// TIA Portal project "project_tia_portal" (V17)

(* hardware
DEVICE "S7-1500/ET200MP station_1"  S7-1500 station
   slot 0: "Rail_0"  Rack  6ES7 590-1***0-0AA0
   slot 1: "PLC_1"  CPU 1513-1 PN  6ES7 513-1AL01-0AB0  V2.6
      slot 3: "CPU display_1"  6ES7591-1AA00-0AA0
      slot 32768: "PROFINET interface_1"  X1
         slot 32769: "Port_1"  X1 P1
         slot 32770: "Port_2"  X1 P2
*)

// ===== PLC "PLC_1"  CPU 1513-1 PN =====

VAR_GLOBAL   // PLC tag table "Default tag table"
   "OPC_START" AT %I0.0 : Bool;
   "OPC_STOP" AT %I0.1 : Bool;
   "SISTEM" AT %M0.0 : Bool;
   "OPC_EMITTER" AT %Q0.0 : Bool;
   "OPC_LONG_BELT" AT %QD2 : Real;
   "OPC_CAPACITIVE_1" AT %I0.2 : Bool;
   "OPC_CAM" AT %QD6 : DInt;
   "OPC_PHOTOELECTRIC" AT %I0.3 : Bool;
   "OPC_GATE_1" AT %Q0.1 : Bool;
   "OPC_GATE_2" AT %Q0.2 : Bool;
   "OPC_PISTON_SENSOR" AT %I0.4 : Bool;
   "OPC_BELT_2" AT %Q0.3 : Bool;
   "OPC_PISTON" AT %QD10 : Real;
   "OPC_CAPACITIVE_2" AT %I0.5 : Bool;
   "ENABLE_BELT_2" AT %M0.5 : Bool;
   "OPC_GATE_FINALE" AT %Q0.4 : Bool;
   "OPC_CAPACITIVE_3" AT %I0.6 : Bool;
   "OPC_X_OUT" AT %QD14 : Real;
   "OPC_Y_OUT" AT %QD18 : Real;
   "OPC_Z_OUT" AT %QD22 : Real;
   "OPC_XY_MOVEMENT" AT %I0.7 : Bool;
   "OPC_Z_MOVEMENT" AT %I1.0 : Bool;
   "OPC_CONFIG" AT %I1.1 : Bool;
   "OPC_EMITTER_2" AT %Q0.5 : Bool;
   "OPC_X_IN" AT %ID2 : Real;
   "OPC_Y_IN" AT %ID6 : Real;
   "OPC_Z_IN" AT %ID10 : Real;
   "OPC_CLAW_BOX_DETECTED" AT %I1.2 : Bool;
   "OPC_CLAW" AT %Q0.6 : Bool;
   "OPC_BELT_LAST_1" AT %Q0.7 : Bool;
   "OPC_BELT_LAST_2" AT %Q1.0 : Bool;
END_VAR

DATA_BLOCK "IEC_Timer_0_DB"   // DB1
{ S7_Optimized_Access := 'TRUE' }
AUTHOR : Simatic
FAMILY : IEC
NAME : IEC_TMR
VERSION : 1.0
// stored: InstanceOfName IEC_TIMER
"IEC_TIMER"
BEGIN
END_DATA_BLOCK

DATA_BLOCK "IEC_Counter_0_DB"   // DB2
{ S7_Optimized_Access := 'TRUE' }
AUTHOR : Simatic
FAMILY : IEC
NAME : CNTR
VERSION : 1.0
// stored: InstanceOfName IEC_COUNTER
"IEC_COUNTER"
BEGIN
END_DATA_BLOCK

DATA_BLOCK "COORDS"   // DB3
{ S7_Optimized_Access := 'TRUE' }
VERSION : 0.1
   VAR
      BOX_X : Real;
      BOX_Y : Real;
      CODE : Int;
      X_LOW : Real;
      X_HIGH : Real;
      Y_LOW : Real;
      Y_HIGH : Real;
      Z_LOW : Real;
      Z_HIGH : Real;
      Y_FINALE : Real;
   END_VAR
BEGIN
END_DATA_BLOCK

DATA_BLOCK "CONFIG_VARS"   // DB7
{ S7_Optimized_Access := 'TRUE' }
VERSION : 0.1
   VAR
      MOVE_2_BOX : Bool;
      Y_POSITION_FINAL : Bool;
      EMITTER_CONFIG : Bool;
      Z_POSITION_FINALE : Bool;
      "COUNTER" : Int;
      TRIG_4_PY_INSTRUCTION : Bool;
      INSTRUCTION_2_PY : Bool;
      PY_RESPONSE : Bool;
      CONFIG_END : Bool;
      TRIG_N : Bool;
      INSTRUCTION_TRIG_N : Bool;
      GATE_FINALE : Bool;
      N_TRIG_FOR_EMITTER : Bool;
      FIRST_MOVE : Bool;
      SECOND_MOV : Bool;
      TRIG_4_MOVE : Bool;
      TRIG_4_2ND_MOVE : Bool;
      TRIG_4_CLAW : Bool;
      TRIG_4_DROP : Bool;
      TRIG_4_RSTART : Bool;
      N_TRIG_FIRST_MOV : Bool;
      N_TRIG_SISTEM : Bool;
   END_VAR
BEGIN
END_DATA_BLOCK

DATA_BLOCK "PRINCIPAL"   // DB8
{ S7_Optimized_Access := 'TRUE' }
VERSION : 0.1
   VAR
      "2_UNITS" : Int;
      N_TRIG_2_UDS : Bool;
      P_TRIG_LONG_BELT : Bool;
      N_TRIG_LONG_BELT : Bool;
      TRIG : Bool;
   END_VAR
BEGIN
END_DATA_BLOCK

DATA_BLOCK "Emitters"   // DB11
{ S7_Optimized_Access := 'TRUE' }
VERSION : 0.1
   VAR
      Trig_1 : Bool;
      Trig_2 : Bool;
      Trig_3 : Bool;
      Trig_4 : Bool;
      Trig_5 : Bool;
   END_VAR
BEGIN
END_DATA_BLOCK

// folder: System blocks/Program resources

DATA_BLOCK "IEC_Timer_0_DB_1"   // DB4
{ S7_Optimized_Access := 'TRUE' }
AUTHOR : Simatic
FAMILY : IEC
NAME : IEC_TMR
VERSION : 1.0
// stored: InstanceOfName IEC_TIMER
"IEC_TIMER"
BEGIN
END_DATA_BLOCK

DATA_BLOCK "IEC_Timer_0_DB_2"   // DB5
{ S7_Optimized_Access := 'TRUE' }
AUTHOR : Simatic
FAMILY : IEC
NAME : IEC_TMR
VERSION : 1.0
// stored: InstanceOfName IEC_TIMER
"IEC_TIMER"
BEGIN
END_DATA_BLOCK

DATA_BLOCK "IEC_Timer_0_DB_3"   // DB6
{ S7_Optimized_Access := 'TRUE' }
AUTHOR : Simatic
FAMILY : IEC
NAME : IEC_TMR
VERSION : 1.0
// stored: InstanceOfName IEC_TIMER
"IEC_TIMER"
BEGIN
END_DATA_BLOCK

DATA_BLOCK "IEC_Timer_0_DB_4"   // DB9
{ S7_Optimized_Access := 'TRUE' }
AUTHOR : Simatic
FAMILY : IEC
NAME : IEC_TMR
VERSION : 1.0
// stored: InstanceOfName IEC_TIMER
"IEC_TIMER"
BEGIN
END_DATA_BLOCK

DATA_BLOCK "IEC_Timer_0_DB_5"   // DB10
{ S7_Optimized_Access := 'TRUE' }
AUTHOR : Simatic
FAMILY : IEC
NAME : IEC_TMR
VERSION : 1.0
// stored: InstanceOfName IEC_TIMER
"IEC_TIMER"
BEGIN
END_DATA_BLOCK

// folder: (top level)

FUNCTION "PICK_PLACE" : Void   // FC2, LAD
{ S7_Optimized_Access := 'TRUE' }
VERSION : 0.1
   VAR_TEMP
      EMITTER_CONFIG : Bool;
      EMITTER_CONFIG_1 : Bool;
      EMITTER_CONFIG_2 : Bool;
   END_VAR
   VAR_TEMP   // added for the SCL form of the ladder/FBD networks
      _w1 : Bool;
      _w2 : Bool;
      _w3 : Bool;
      _w4 : Bool;
      _w5 : Bool;
      _w6 : Bool;
   END_VAR
BEGIN

REGION Network 1
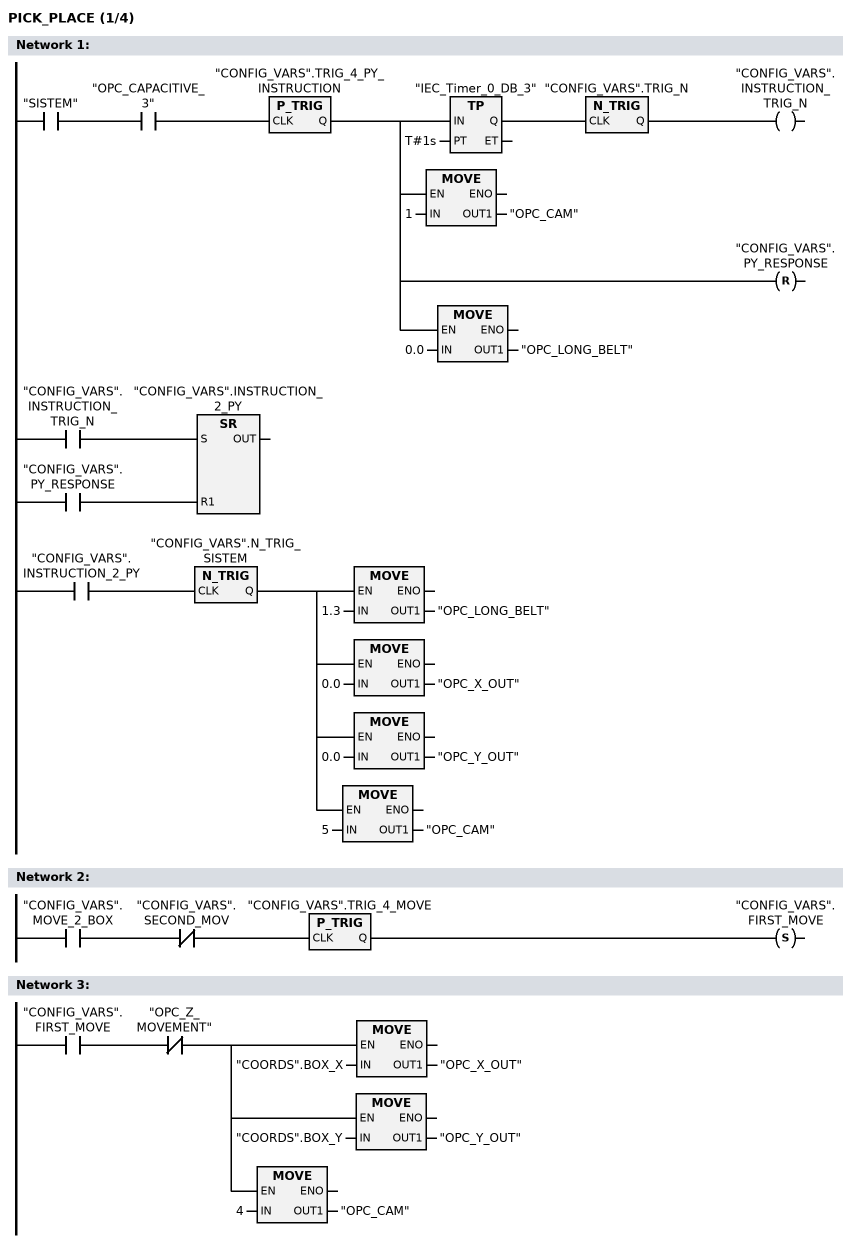
   #_w1 := "SISTEM" AND "OPC_CAPACITIVE_3";
   #_w2 := #_w1 AND NOT "CONFIG_VARS".TRIG_4_PY_INSTRUCTION;   // rising edge
   "CONFIG_VARS".TRIG_4_PY_INSTRUCTION := #_w1;
   "IEC_Timer_0_DB_3".TP(IN := #_w2, PT := T#1s);
   #_w3 := NOT "IEC_Timer_0_DB_3".Q AND "CONFIG_VARS".TRIG_N;   // falling edge
   "CONFIG_VARS".TRIG_N := "IEC_Timer_0_DB_3".Q;
   "CONFIG_VARS".INSTRUCTION_TRIG_N := #_w3;
   IF #_w2 THEN
       "OPC_CAM" := 1;
       "CONFIG_VARS".PY_RESPONSE := FALSE;
       "OPC_LONG_BELT" := 0.0;
   END_IF;
   IF "CONFIG_VARS".INSTRUCTION_TRIG_N THEN
       "CONFIG_VARS".INSTRUCTION_2_PY := TRUE;   // SR flip-flop
   END_IF;
   IF "CONFIG_VARS".PY_RESPONSE THEN "CONFIG_VARS".INSTRUCTION_2_PY := FALSE; END_IF;
   #_w4 := NOT "CONFIG_VARS".INSTRUCTION_2_PY AND "CONFIG_VARS".N_TRIG_SISTEM;   // falling edge
   "CONFIG_VARS".N_TRIG_SISTEM := "CONFIG_VARS".INSTRUCTION_2_PY;
   IF #_w4 THEN
       "OPC_LONG_BELT" := 1.3;
       "OPC_X_OUT" := 0.0;
       "OPC_Y_OUT" := 0.0;
       "OPC_CAM" := 5;
   END_IF;
END_REGION

REGION Network 2
   RUNG wire#powerrail
      Contact( "CONFIG_VARS".MOVE_2_BOX )
      I_Contact( "CONFIG_VARS".SECOND_MOV )
      P_Trig( "CONFIG_VARS".TRIG_4_MOVE )
      S_Coil( "CONFIG_VARS".FIRST_MOVE )
   END_RUNG
   // the same network as SCL:
   #_w1 := "CONFIG_VARS".MOVE_2_BOX AND NOT "CONFIG_VARS".SECOND_MOV;
   #_w2 := #_w1 AND NOT "CONFIG_VARS".TRIG_4_MOVE;   // rising edge
   "CONFIG_VARS".TRIG_4_MOVE := #_w1;
   IF #_w2 THEN "CONFIG_VARS".FIRST_MOVE := TRUE; END_IF;
END_REGION

REGION Network 3
   RUNG wire#powerrail
      Contact( "CONFIG_VARS".FIRST_MOVE )
      I_Contact( "OPC_Z_MOVEMENT" )
      wire#w1
      Move(in := "COORDS".BOX_X, out1 => "OPC_X_OUT")
   END_RUNG
   RUNG wire#w1
      Move(in := "COORDS".BOX_Y, out1 => "OPC_Y_OUT")
   END_RUNG
   RUNG wire#w1
      Move(in := 4, out1 => "OPC_CAM")
   END_RUNG
   // the same network as SCL:
   IF "CONFIG_VARS".FIRST_MOVE AND NOT "OPC_Z_MOVEMENT" THEN
       "OPC_X_OUT" := "COORDS".BOX_X;
       "OPC_Y_OUT" := "COORDS".BOX_Y;
       "OPC_CAM" := 4;
   END_IF;
END_REGION

REGION Network 4
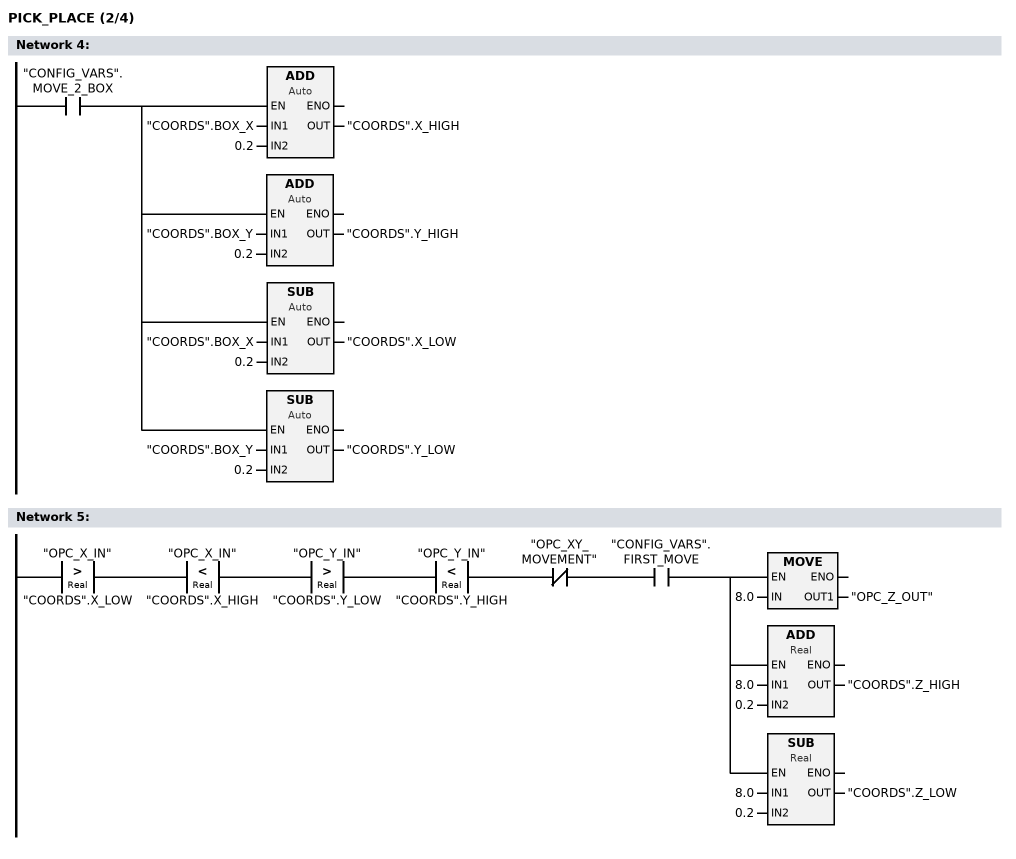
   RUNG wire#powerrail
      Contact( "CONFIG_VARS".MOVE_2_BOX )
      wire#w1
      Add(in1 := "COORDS".BOX_X, in2 := 0.2, out => "COORDS".X_HIGH)
   END_RUNG
   RUNG wire#w1
      Add(in1 := "COORDS".BOX_Y, in2 := 0.2, out => "COORDS".Y_HIGH)
   END_RUNG
   RUNG wire#w1
      Sub(in1 := "COORDS".BOX_X, in2 := 0.2, out => "COORDS".X_LOW)
   END_RUNG
   RUNG wire#w1
      Sub(in1 := "COORDS".BOX_Y, in2 := 0.2, out => "COORDS".Y_LOW)
   END_RUNG
   // the same network as SCL:
   IF "CONFIG_VARS".MOVE_2_BOX THEN
       "COORDS".X_HIGH := "COORDS".BOX_X + 0.2;
       "COORDS".Y_HIGH := "COORDS".BOX_Y + 0.2;
       "COORDS".X_LOW := "COORDS".BOX_X - 0.2;
       "COORDS".Y_LOW := "COORDS".BOX_Y - 0.2;
   END_IF;
END_REGION

REGION Network 5
   RUNG wire#powerrail
      { S7_Templates := "SrcType := Real" } GT_Contact(in1 := "OPC_X_IN", in2 := "COORDS".X_LOW)
      { S7_Templates := "SrcType := Real" } LT_Contact(in1 := "OPC_X_IN", in2 := "COORDS".X_HIGH)
      { S7_Templates := "SrcType := Real" } GT_Contact(in1 := "OPC_Y_IN", in2 := "COORDS".Y_LOW)
      { S7_Templates := "SrcType := Real" } LT_Contact(in1 := "OPC_Y_IN", in2 := "COORDS".Y_HIGH)
      I_Contact( "OPC_XY_MOVEMENT" )
      Contact( "CONFIG_VARS".FIRST_MOVE )
      wire#w1
      Move(in := 8.0, out1 => "OPC_Z_OUT")
   END_RUNG
   RUNG wire#w1
      { S7_Templates := "SrcType := Real" } Add(in1 := 8.0, in2 := 0.2, out => "COORDS".Z_HIGH)
   END_RUNG
   RUNG wire#w1
      { S7_Templates := "SrcType := Real" } Sub(in1 := 8.0, in2 := 0.2, out => "COORDS".Z_LOW)
   END_RUNG
   // the same network as SCL:
   IF ("OPC_X_IN" > "COORDS".X_LOW) AND ("OPC_X_IN" < "COORDS".X_HIGH) AND ("OPC_Y_IN" > "COORDS".Y_LOW) AND ("OPC_Y_IN" < "COORDS".Y_HIGH) AND NOT "OPC_XY_MOVEMENT" AND "CONFIG_VARS".FIRST_MOVE THEN
       "OPC_Z_OUT" := 8.0;
       "COORDS".Z_HIGH := 8.0 + 0.2;
       "COORDS".Z_LOW := 8.0 - 0.2;
   END_IF;
END_REGION

REGION Network 6
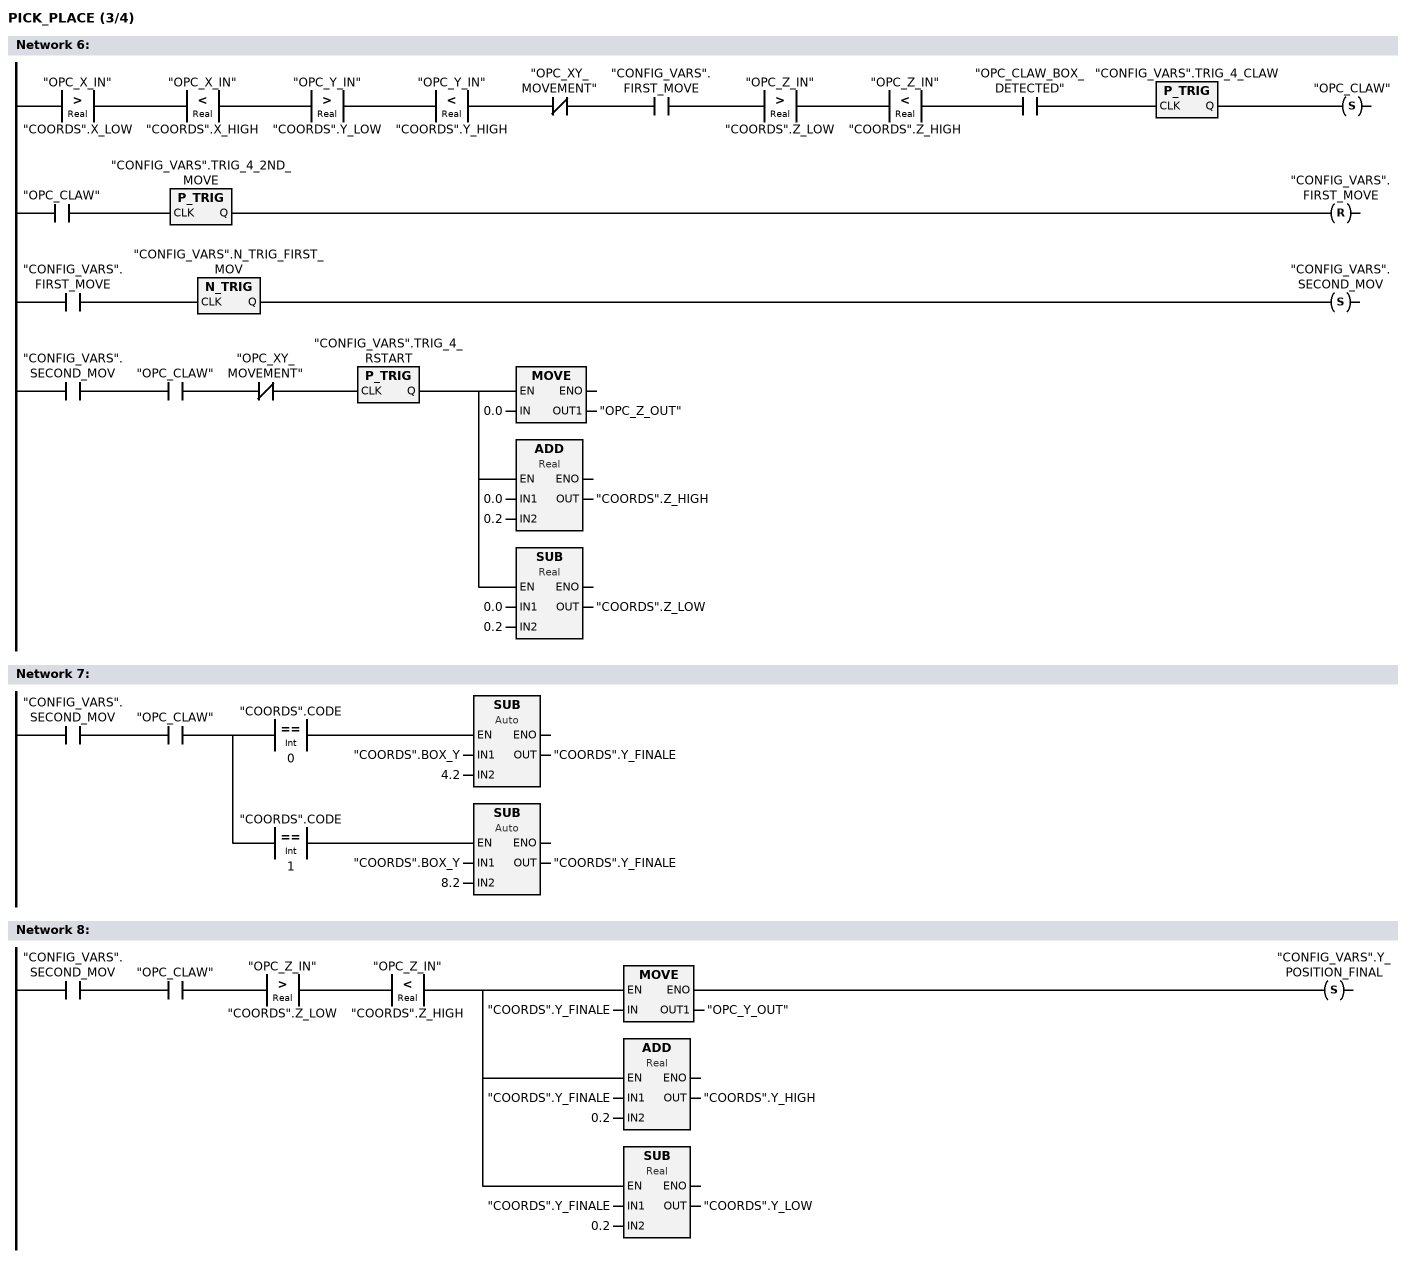
   RUNG wire#powerrail
      { S7_Templates := "SrcType := Real" } GT_Contact(in1 := "OPC_X_IN", in2 := "COORDS".X_LOW)
      { S7_Templates := "SrcType := Real" } LT_Contact(in1 := "OPC_X_IN", in2 := "COORDS".X_HIGH)
      { S7_Templates := "SrcType := Real" } GT_Contact(in1 := "OPC_Y_IN", in2 := "COORDS".Y_LOW)
      { S7_Templates := "SrcType := Real" } LT_Contact(in1 := "OPC_Y_IN", in2 := "COORDS".Y_HIGH)
      I_Contact( "OPC_XY_MOVEMENT" )
      Contact( "CONFIG_VARS".FIRST_MOVE )
      { S7_Templates := "SrcType := Real" } GT_Contact(in1 := "OPC_Z_IN", in2 := "COORDS".Z_LOW)
      { S7_Templates := "SrcType := Real" } LT_Contact(in1 := "OPC_Z_IN", in2 := "COORDS".Z_HIGH)
      Contact( "OPC_CLAW_BOX_DETECTED" )
      P_Trig( "CONFIG_VARS".TRIG_4_CLAW )
      S_Coil( "OPC_CLAW" )
   END_RUNG
   RUNG wire#powerrail
      Contact( "OPC_CLAW" )
      P_Trig( "CONFIG_VARS".TRIG_4_2ND_MOVE )
      R_Coil( "CONFIG_VARS".FIRST_MOVE )
   END_RUNG
   RUNG wire#powerrail
      Contact( "CONFIG_VARS".FIRST_MOVE )
      N_Trig( "CONFIG_VARS".N_TRIG_FIRST_MOV )
      S_Coil( "CONFIG_VARS".SECOND_MOV )
   END_RUNG
   RUNG wire#powerrail
      Contact( "CONFIG_VARS".SECOND_MOV )
      Contact( "OPC_CLAW" )
      I_Contact( "OPC_XY_MOVEMENT" )
      P_Trig( "CONFIG_VARS".TRIG_4_RSTART )
      wire#w1
      Move(in := 0.0, out1 => "OPC_Z_OUT")
   END_RUNG
   RUNG wire#w1
      { S7_Templates := "SrcType := Real" } Add(in1 := 0.0, in2 := 0.2, out => "COORDS".Z_HIGH)
   END_RUNG
   RUNG wire#w1
      { S7_Templates := "SrcType := Real" } Sub(in1 := 0.0, in2 := 0.2, out => "COORDS".Z_LOW)
   END_RUNG
   // the same network as SCL:
   #_w1 := ("OPC_X_IN" > "COORDS".X_LOW) AND ("OPC_X_IN" < "COORDS".X_HIGH) AND ("OPC_Y_IN" > "COORDS".Y_LOW) AND ("OPC_Y_IN" < "COORDS".Y_HIGH) AND NOT "OPC_XY_MOVEMENT" AND "CONFIG_VARS".FIRST_MOVE AND ("OPC_Z_IN" > "COORDS".Z_LOW) AND ("OPC_Z_IN" < "COORDS".Z_HIGH) AND "OPC_CLAW_BOX_DETECTED";
   #_w2 := #_w1 AND NOT "CONFIG_VARS".TRIG_4_CLAW;   // rising edge
   "CONFIG_VARS".TRIG_4_CLAW := #_w1;
   IF #_w2 THEN "OPC_CLAW" := TRUE; END_IF;
   #_w3 := "OPC_CLAW" AND NOT "CONFIG_VARS".TRIG_4_2ND_MOVE;   // rising edge
   "CONFIG_VARS".TRIG_4_2ND_MOVE := "OPC_CLAW";
   IF #_w3 THEN "CONFIG_VARS".FIRST_MOVE := FALSE; END_IF;
   #_w4 := NOT "CONFIG_VARS".FIRST_MOVE AND "CONFIG_VARS".N_TRIG_FIRST_MOV;   // falling edge
   "CONFIG_VARS".N_TRIG_FIRST_MOV := "CONFIG_VARS".FIRST_MOVE;
   IF #_w4 THEN "CONFIG_VARS".SECOND_MOV := TRUE; END_IF;
   #_w5 := "CONFIG_VARS".SECOND_MOV AND "OPC_CLAW" AND NOT "OPC_XY_MOVEMENT";
   #_w6 := #_w5 AND NOT "CONFIG_VARS".TRIG_4_RSTART;   // rising edge
   "CONFIG_VARS".TRIG_4_RSTART := #_w5;
   IF #_w6 THEN
       "OPC_Z_OUT" := 0.0;
       "COORDS".Z_HIGH := 0.0 + 0.2;
       "COORDS".Z_LOW := 0.0 - 0.2;
   END_IF;
END_REGION

REGION Network 7
   RUNG wire#powerrail
      Contact( "CONFIG_VARS".SECOND_MOV )
      Contact( "OPC_CLAW" )
      wire#w1
      { S7_Templates := "SrcType := Int" } EQ_Contact(in1 := "COORDS".CODE, in2 := 0)
      Sub(in1 := "COORDS".BOX_Y, in2 := 4.2, out => "COORDS".Y_FINALE)
   END_RUNG
   RUNG wire#w1
      { S7_Templates := "SrcType := Int" } EQ_Contact(in1 := "COORDS".CODE, in2 := 1)
      Sub(in1 := "COORDS".BOX_Y, in2 := 8.2, out => "COORDS".Y_FINALE)
   END_RUNG
   // the same network as SCL:
   #_w1 := "CONFIG_VARS".SECOND_MOV AND "OPC_CLAW";
   IF #_w1 AND ("COORDS".CODE = 0) THEN "COORDS".Y_FINALE := "COORDS".BOX_Y - 4.2; END_IF;
   IF #_w1 AND ("COORDS".CODE = 1) THEN "COORDS".Y_FINALE := "COORDS".BOX_Y - 8.2; END_IF;
END_REGION

REGION Network 8
   RUNG wire#powerrail
      Contact( "CONFIG_VARS".SECOND_MOV )
      Contact( "OPC_CLAW" )
      { S7_Templates := "SrcType := Real" } GT_Contact(in1 := "OPC_Z_IN", in2 := "COORDS".Z_LOW)
      { S7_Templates := "SrcType := Real" } LT_Contact(in1 := "OPC_Z_IN", in2 := "COORDS".Z_HIGH)
      wire#w1
      Move(in := "COORDS".Y_FINALE, out1 => "OPC_Y_OUT")
      S_Coil( "CONFIG_VARS".Y_POSITION_FINAL )
   END_RUNG
   RUNG wire#w1
      { S7_Templates := "SrcType := Real" } Add(in1 := "COORDS".Y_FINALE, in2 := 0.2, out => "COORDS".Y_HIGH)
   END_RUNG
   RUNG wire#w1
      { S7_Templates := "SrcType := Real" } Sub(in1 := "COORDS".Y_FINALE, in2 := 0.2, out => "COORDS".Y_LOW)
   END_RUNG
   // the same network as SCL:
   IF "CONFIG_VARS".SECOND_MOV AND "OPC_CLAW" AND ("OPC_Z_IN" > "COORDS".Z_LOW) AND ("OPC_Z_IN" < "COORDS".Z_HIGH) THEN
       "OPC_Y_OUT" := "COORDS".Y_FINALE;
       "CONFIG_VARS".Y_POSITION_FINAL := TRUE;
       "COORDS".Y_HIGH := "COORDS".Y_FINALE + 0.2;
       "COORDS".Y_LOW := "COORDS".Y_FINALE - 0.2;
   END_IF;
END_REGION

REGION Network 9
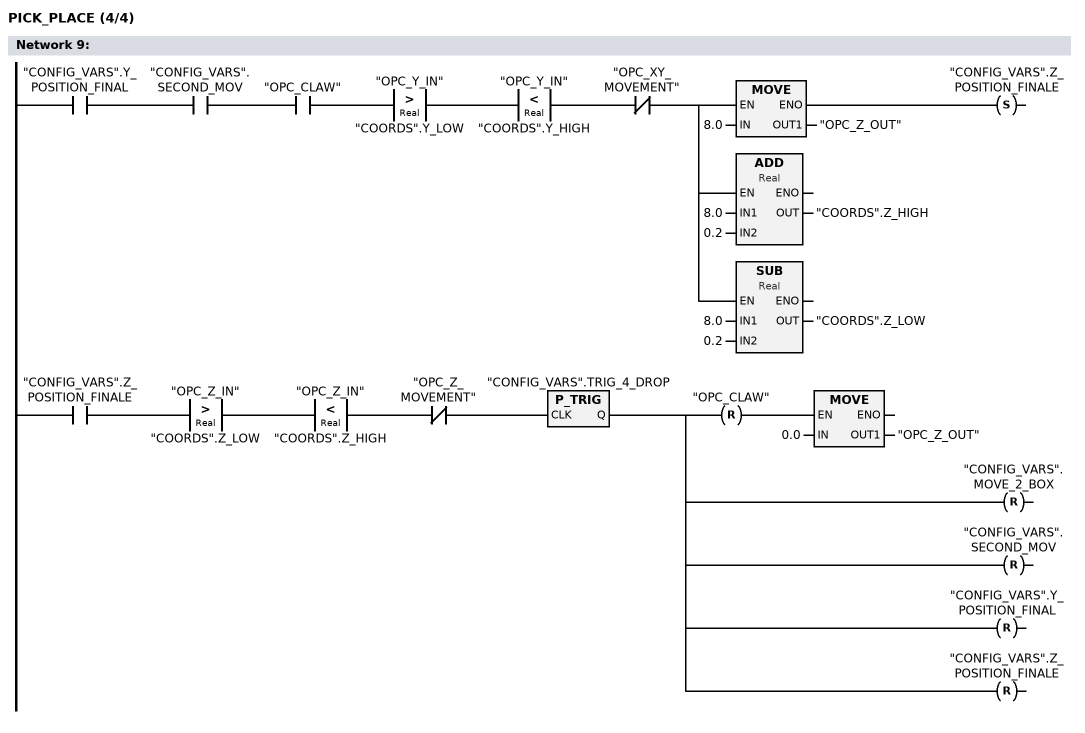
   RUNG wire#powerrail
      Contact( "CONFIG_VARS".Y_POSITION_FINAL )
      Contact( "CONFIG_VARS".SECOND_MOV )
      Contact( "OPC_CLAW" )
      { S7_Templates := "SrcType := Real" } GT_Contact(in1 := "OPC_Y_IN", in2 := "COORDS".Y_LOW)
      { S7_Templates := "SrcType := Real" } LT_Contact(in1 := "OPC_Y_IN", in2 := "COORDS".Y_HIGH)
      I_Contact( "OPC_XY_MOVEMENT" )
      wire#w1
      Move(in := 8.0, out1 => "OPC_Z_OUT")
      S_Coil( "CONFIG_VARS".Z_POSITION_FINALE )
   END_RUNG
   RUNG wire#w1
      { S7_Templates := "SrcType := Real" } Add(in1 := 8.0, in2 := 0.2, out => "COORDS".Z_HIGH)
   END_RUNG
   RUNG wire#w1
      { S7_Templates := "SrcType := Real" } Sub(in1 := 8.0, in2 := 0.2, out => "COORDS".Z_LOW)
   END_RUNG
   RUNG wire#powerrail
      Contact( "CONFIG_VARS".Z_POSITION_FINALE )
      { S7_Templates := "SrcType := Real" } GT_Contact(in1 := "OPC_Z_IN", in2 := "COORDS".Z_LOW)
      { S7_Templates := "SrcType := Real" } LT_Contact(in1 := "OPC_Z_IN", in2 := "COORDS".Z_HIGH)
      I_Contact( "OPC_Z_MOVEMENT" )
      P_Trig( "CONFIG_VARS".TRIG_4_DROP )
      wire#w2
      R_Coil( "OPC_CLAW" )
      Move(in := 0.0, out1 => "OPC_Z_OUT")
   END_RUNG
   RUNG wire#w2
      R_Coil( "CONFIG_VARS".MOVE_2_BOX )
   END_RUNG
   RUNG wire#w2
      R_Coil( "CONFIG_VARS".SECOND_MOV )
   END_RUNG
   RUNG wire#w2
      R_Coil( "CONFIG_VARS".Y_POSITION_FINAL )
   END_RUNG
   RUNG wire#w2
      R_Coil( "CONFIG_VARS".Z_POSITION_FINALE )
   END_RUNG
   // the same network as SCL:
   IF "CONFIG_VARS".Y_POSITION_FINAL AND "CONFIG_VARS".SECOND_MOV AND "OPC_CLAW" AND ("OPC_Y_IN" > "COORDS".Y_LOW) AND ("OPC_Y_IN" < "COORDS".Y_HIGH) AND NOT "OPC_XY_MOVEMENT" THEN
       "OPC_Z_OUT" := 8.0;
       "CONFIG_VARS".Z_POSITION_FINALE := TRUE;
       "COORDS".Z_HIGH := 8.0 + 0.2;
       "COORDS".Z_LOW := 8.0 - 0.2;
   END_IF;
   #_w1 := "CONFIG_VARS".Z_POSITION_FINALE AND ("OPC_Z_IN" > "COORDS".Z_LOW) AND ("OPC_Z_IN" < "COORDS".Z_HIGH) AND NOT "OPC_Z_MOVEMENT";
   #_w2 := #_w1 AND NOT "CONFIG_VARS".TRIG_4_DROP;   // rising edge
   "CONFIG_VARS".TRIG_4_DROP := #_w1;
   IF #_w2 THEN
       "OPC_CLAW" := FALSE;
       "OPC_Z_OUT" := 0.0;
       "CONFIG_VARS".MOVE_2_BOX := FALSE;
       "CONFIG_VARS".SECOND_MOV := FALSE;
       "CONFIG_VARS".Y_POSITION_FINAL := FALSE;
       "CONFIG_VARS".Z_POSITION_FINALE := FALSE;
   END_IF;
END_REGION
END_FUNCTION

ORGANIZATION_BLOCK "Main"   // OB1, LAD, ProgramCycle
TITLE = "Main Program Sweep (Cycle)"
{ S7_Optimized_Access := 'TRUE' }
VERSION : 0.1
   VAR_INPUT
      Initial_Call : Bool;   // Initial call of this OB
      Remanence : Bool;   // =True, if remanent data are available
   END_VAR
   VAR_TEMP   // added for the SCL form of the ladder/FBD networks
      _w1 : Bool;
      _w2 : Bool;
      _w3 : Bool;
      _w4 : Bool;
      _w5 : Bool;
      _w6 : Bool;
   END_VAR
BEGIN

REGION Network 1: Arranque y parada del proceso
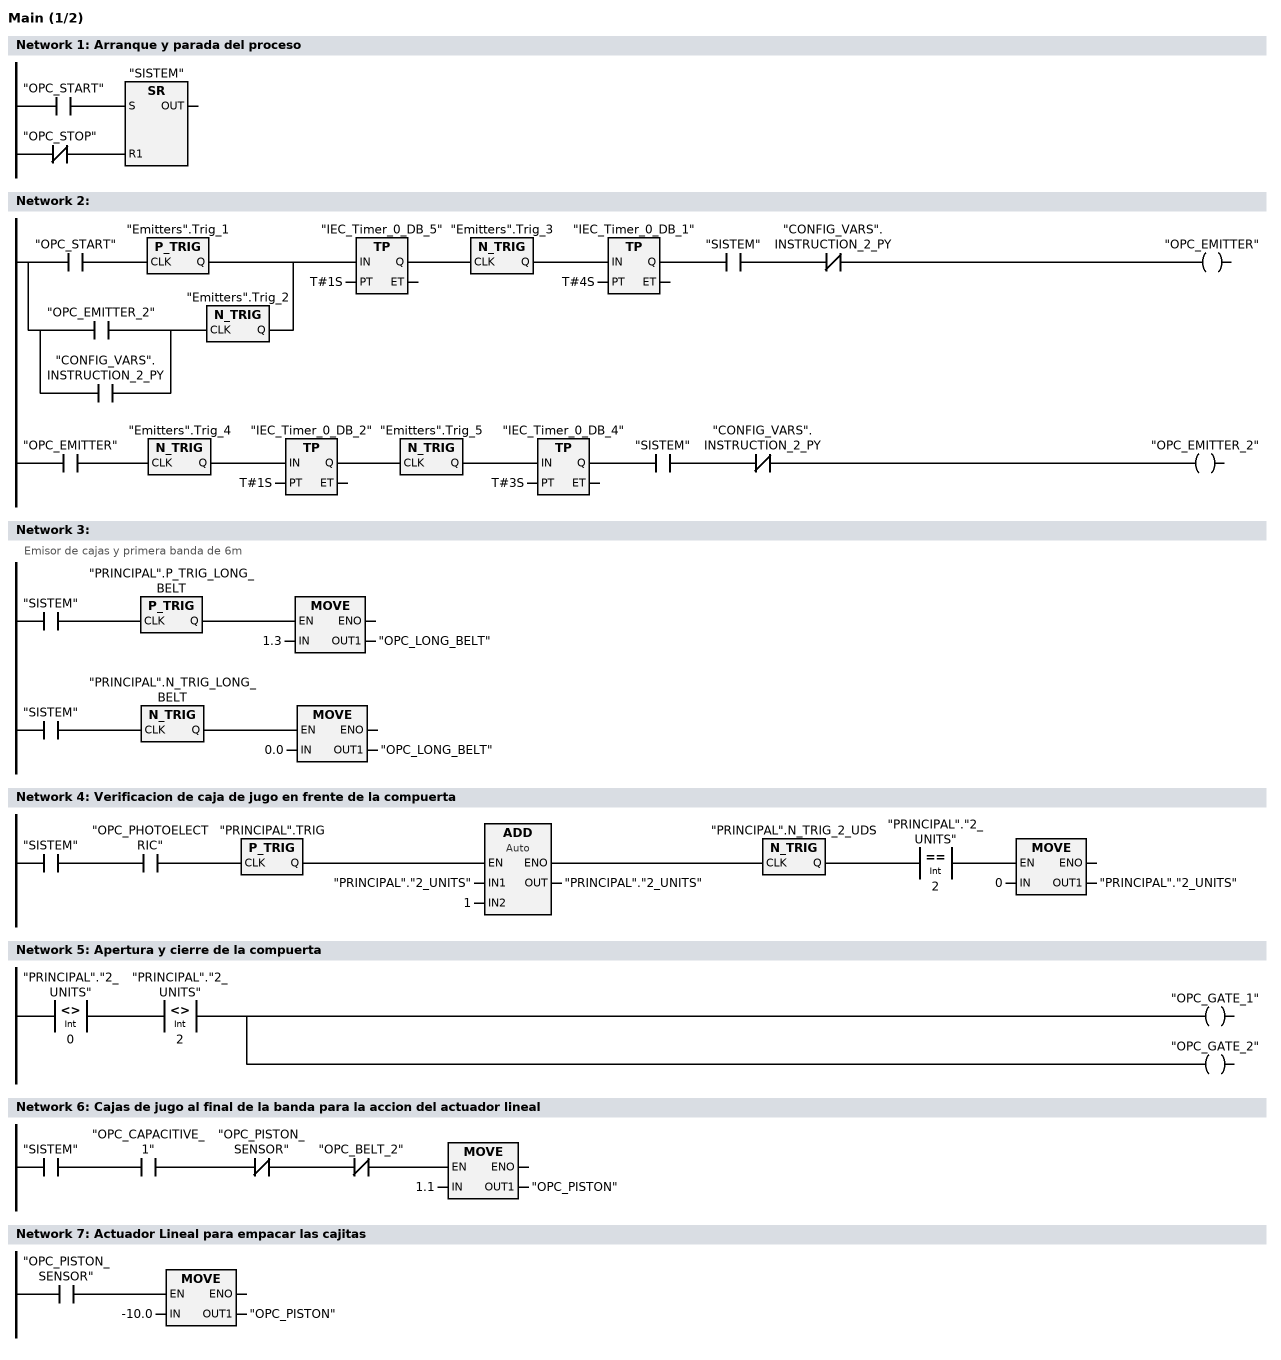
   RUNG wire#powerrail
      Contact( "OPC_START" )
      S_SR(operand := "SISTEM", r1 := wire#w1)
   END_RUNG
   RUNG wire#powerrail
      I_Contact( "OPC_STOP" )
   END_RUNG wire#w1
   // the same network as SCL:
   IF "OPC_START" THEN
       "SISTEM" := TRUE;   // SR flip-flop
   END_IF;
   IF NOT "OPC_STOP" THEN "SISTEM" := FALSE; END_IF;
END_REGION

REGION Network 2
   #_w1 := "OPC_START" AND NOT "Emitters".Trig_1;   // rising edge
   "Emitters".Trig_1 := "OPC_START";
   #_w2 := "OPC_EMITTER_2" OR "CONFIG_VARS".INSTRUCTION_2_PY;
   #_w3 := NOT #_w2 AND "Emitters".Trig_2;   // falling edge
   "Emitters".Trig_2 := #_w2;
   "IEC_Timer_0_DB_5".TP(IN := #_w1 OR #_w3, PT := T#1S);
   #_w4 := NOT "IEC_Timer_0_DB_5".Q AND "Emitters".Trig_3;   // falling edge
   "Emitters".Trig_3 := "IEC_Timer_0_DB_5".Q;
   "IEC_Timer_0_DB_1".TP(IN := #_w4, PT := T#4S);
   "OPC_EMITTER" := "IEC_Timer_0_DB_1".Q AND "SISTEM" AND NOT "CONFIG_VARS".INSTRUCTION_2_PY;
   #_w5 := NOT "OPC_EMITTER" AND "Emitters".Trig_4;   // falling edge
   "Emitters".Trig_4 := "OPC_EMITTER";
   "IEC_Timer_0_DB_2".TP(IN := #_w5, PT := T#1S);
   #_w6 := NOT "IEC_Timer_0_DB_2".Q AND "Emitters".Trig_5;   // falling edge
   "Emitters".Trig_5 := "IEC_Timer_0_DB_2".Q;
   "IEC_Timer_0_DB_4".TP(IN := #_w6, PT := T#3S);
   "OPC_EMITTER_2" := "IEC_Timer_0_DB_4".Q AND "SISTEM" AND NOT "CONFIG_VARS".INSTRUCTION_2_PY;
END_REGION

REGION Network 3
   // Emisor de cajas y primera banda de 6m
   RUNG wire#powerrail
      Contact( "SISTEM" )
      P_Trig( "PRINCIPAL".P_TRIG_LONG_BELT )
      Move(in := 1.3, out1 => "OPC_LONG_BELT")
   END_RUNG
   RUNG wire#powerrail
      Contact( "SISTEM" )
      N_Trig( "PRINCIPAL".N_TRIG_LONG_BELT )
      Move(in := 0.0, out1 => "OPC_LONG_BELT")
   END_RUNG
   // the same network as SCL:
   #_w1 := "SISTEM" AND NOT "PRINCIPAL".P_TRIG_LONG_BELT;   // rising edge
   "PRINCIPAL".P_TRIG_LONG_BELT := "SISTEM";
   IF #_w1 THEN "OPC_LONG_BELT" := 1.3; END_IF;
   #_w2 := NOT "SISTEM" AND "PRINCIPAL".N_TRIG_LONG_BELT;   // falling edge
   "PRINCIPAL".N_TRIG_LONG_BELT := "SISTEM";
   IF #_w2 THEN "OPC_LONG_BELT" := 0.0; END_IF;
END_REGION

REGION Network 4: Verificacion de caja de jugo en frente de la compuerta
   RUNG wire#powerrail
      Contact( "SISTEM" )
      Contact( "OPC_PHOTOELECTRIC" )
      P_Trig( "PRINCIPAL".TRIG )
      Add(in1 := "PRINCIPAL"."2_UNITS", in2 := 1, out => "PRINCIPAL"."2_UNITS")
      N_Trig( "PRINCIPAL".N_TRIG_2_UDS )
      { S7_Templates := "SrcType := Int" } EQ_Contact(in1 := "PRINCIPAL"."2_UNITS", in2 := 2)
      Move(in := 0, out1 => "PRINCIPAL"."2_UNITS")
   END_RUNG
   // the same network as SCL:
   #_w1 := "SISTEM" AND "OPC_PHOTOELECTRIC";
   #_w2 := #_w1 AND NOT "PRINCIPAL".TRIG;   // rising edge
   "PRINCIPAL".TRIG := #_w1;
   IF #_w2 THEN "PRINCIPAL"."2_UNITS" := "PRINCIPAL"."2_UNITS" + 1; END_IF;
   #_w3 := NOT #_w2 AND "PRINCIPAL".N_TRIG_2_UDS;   // falling edge
   "PRINCIPAL".N_TRIG_2_UDS := #_w2;
   IF #_w3 AND ("PRINCIPAL"."2_UNITS" = 2) THEN "PRINCIPAL"."2_UNITS" := 0; END_IF;
END_REGION

REGION Network 5: Apertura y cierre de la compuerta
   RUNG wire#powerrail
      { S7_Templates := "SrcType := Int" } NE_Contact(in1 := "PRINCIPAL"."2_UNITS", in2 := 0)
      { S7_Templates := "SrcType := Int" } NE_Contact(in1 := "PRINCIPAL"."2_UNITS", in2 := 2)
      wire#w1
      Coil( "OPC_GATE_1" )
   END_RUNG
   RUNG wire#w1
      Coil( "OPC_GATE_2" )
   END_RUNG
   // the same network as SCL:
   "OPC_GATE_1" := ("PRINCIPAL"."2_UNITS" <> 0) AND ("PRINCIPAL"."2_UNITS" <> 2);
   "OPC_GATE_2" := "OPC_GATE_1";
END_REGION

REGION Network 6: Cajas de jugo al final de la banda para la accion del actuador lineal
   RUNG wire#powerrail
      Contact( "SISTEM" )
      Contact( "OPC_CAPACITIVE_1" )
      I_Contact( "OPC_PISTON_SENSOR" )
      I_Contact( "OPC_BELT_2" )
      Move(in := 1.1, out1 => "OPC_PISTON")
   END_RUNG
   // the same network as SCL:
   IF "SISTEM" AND "OPC_CAPACITIVE_1" AND NOT "OPC_PISTON_SENSOR" AND NOT "OPC_BELT_2" THEN
       "OPC_PISTON" := 1.1;
   END_IF;
END_REGION

REGION Network 7: Actuador Lineal para empacar las cajitas
   RUNG wire#powerrail
      Contact( "OPC_PISTON_SENSOR" )
      Move(in := -10.0, out1 => "OPC_PISTON")
   END_RUNG
   // the same network as SCL:
   IF "OPC_PISTON_SENSOR" THEN "OPC_PISTON" := -10.0; END_IF;
END_REGION

REGION Network 8
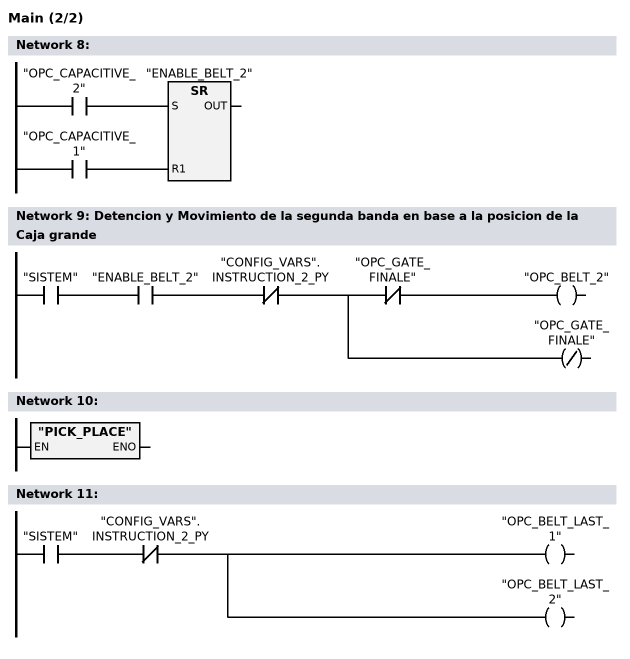
   RUNG wire#powerrail
      Contact( "OPC_CAPACITIVE_2" )
      S_SR(operand := "ENABLE_BELT_2", r1 := wire#w1)
   END_RUNG
   RUNG wire#powerrail
      Contact( "OPC_CAPACITIVE_1" )
   END_RUNG wire#w1
   // the same network as SCL:
   IF "OPC_CAPACITIVE_2" THEN
       "ENABLE_BELT_2" := TRUE;   // SR flip-flop
   END_IF;
   IF "OPC_CAPACITIVE_1" THEN "ENABLE_BELT_2" := FALSE; END_IF;
END_REGION

REGION Network 9: Detencion y Movimiento de la segunda banda en base a la posicion de la Caja grande
   RUNG wire#powerrail
      Contact( "SISTEM" )
      Contact( "ENABLE_BELT_2" )
      I_Contact( "CONFIG_VARS".INSTRUCTION_2_PY )
      wire#w1
      I_Contact( "OPC_GATE_FINALE" )
      Coil( "OPC_BELT_2" )
   END_RUNG
   RUNG wire#w1
      I_Coil( "OPC_GATE_FINALE" )
   END_RUNG
   // the same network as SCL:
   #_w1 := "SISTEM" AND "ENABLE_BELT_2" AND NOT "CONFIG_VARS".INSTRUCTION_2_PY;
   "OPC_BELT_2" := #_w1 AND NOT "OPC_GATE_FINALE";
   "OPC_GATE_FINALE" := NOT #_w1;
END_REGION

REGION Network 10
   RUNG wire#powerrail
      "PICK_PLACE"()
   END_RUNG
   // the same network as SCL:
   "PICK_PLACE"();
END_REGION

REGION Network 11
   RUNG wire#powerrail
      Contact( "SISTEM" )
      I_Contact( "CONFIG_VARS".INSTRUCTION_2_PY )
      wire#w1
      Coil( "OPC_BELT_LAST_1" )
   END_RUNG
   RUNG wire#w1
      Coil( "OPC_BELT_LAST_2" )
   END_RUNG
   // the same network as SCL:
   "OPC_BELT_LAST_1" := "SISTEM" AND NOT "CONFIG_VARS".INSTRUCTION_2_PY;
   "OPC_BELT_LAST_2" := "OPC_BELT_LAST_1";
END_REGION
END_ORGANIZATION_BLOCK